// TIA Portal V20 export
FUNCTION "Safety Door" : Void   // FC97, LAD
// stored: SetENOAutomatically false
   VAR CONSTANT
      TRUE : Bool := TRUE;
      FALSE : Bool;
   END_VAR
   VAR_TEMP   // added for the SCL form of the ladder/FBD networks
      _w1 : Bool;
   END_VAR
BEGIN

REGION Network 1: FDoorEC.TOP Monitoring
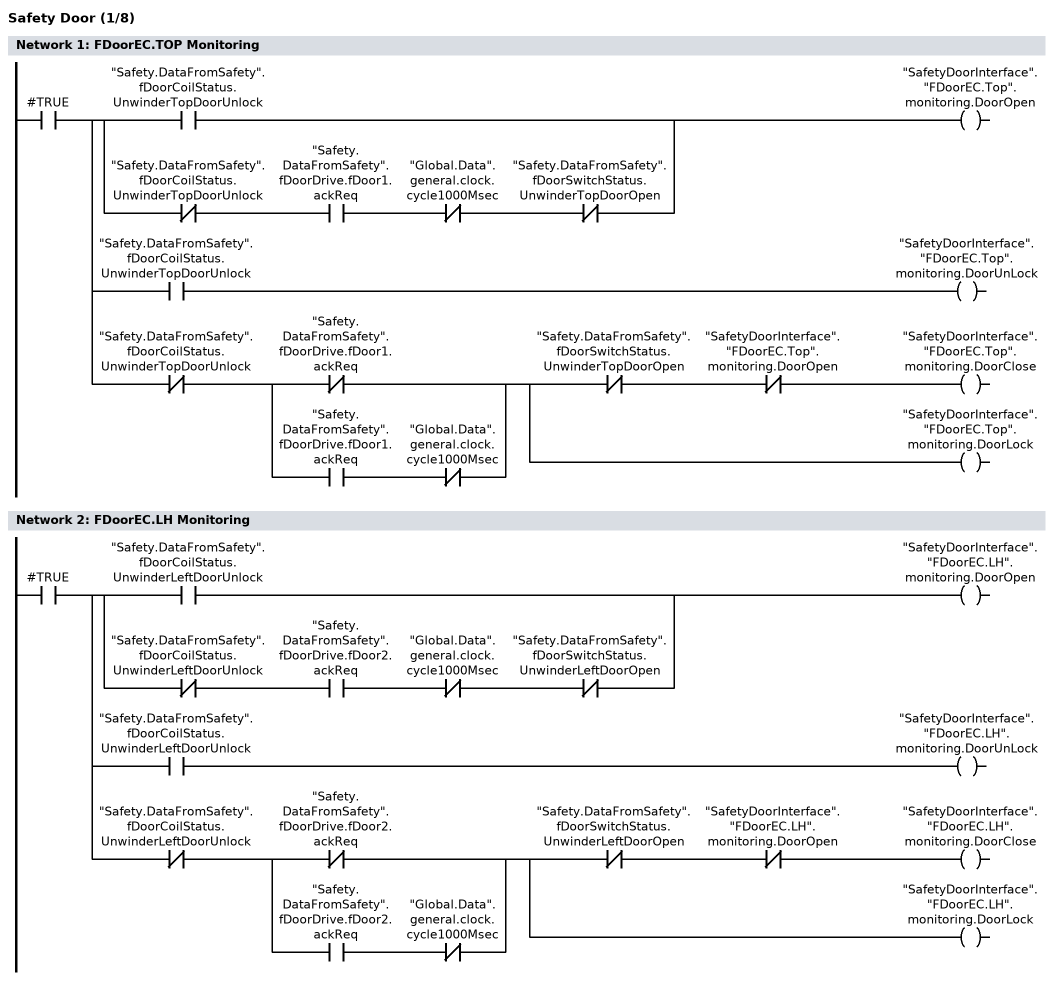
   RUNG wire#powerrail
      Contact( #TRUE )
      wire#w1
      Contact( "Safety.DataFromSafety".fDoorCoilStatus.UnwinderTopDoorUnlock )
      wire#w2
      Coil( "SafetyDoorInterface"."FDoorEC.Top".monitoring.DoorOpen )
   END_RUNG
   RUNG wire#w1
      I_Contact( "Safety.DataFromSafety".fDoorCoilStatus.UnwinderTopDoorUnlock )
      Contact( "Safety.DataFromSafety".fDoorDrive.fDoor1.ackReq )
      I_Contact( "Global.Data".general.clock.cycle1000Msec )
      I_Contact( "Safety.DataFromSafety".fDoorSwitchStatus.UnwinderTopDoorOpen )
   END_RUNG wire#w2
   RUNG wire#w1
      Contact( "Safety.DataFromSafety".fDoorCoilStatus.UnwinderTopDoorUnlock )
      Coil( "SafetyDoorInterface"."FDoorEC.Top".monitoring.DoorUnLock )
   END_RUNG
   RUNG wire#w1
      I_Contact( "Safety.DataFromSafety".fDoorCoilStatus.UnwinderTopDoorUnlock )
      wire#w3
      I_Contact( "Safety.DataFromSafety".fDoorDrive.fDoor1.ackReq )
      wire#w4
      I_Contact( "Safety.DataFromSafety".fDoorSwitchStatus.UnwinderTopDoorOpen )
      I_Contact( "SafetyDoorInterface"."FDoorEC.Top".monitoring.DoorOpen )
      Coil( "SafetyDoorInterface"."FDoorEC.Top".monitoring.DoorClose )
   END_RUNG
   RUNG wire#w3
      Contact( "Safety.DataFromSafety".fDoorDrive.fDoor1.ackReq )
      I_Contact( "Global.Data".general.clock.cycle1000Msec )
   END_RUNG wire#w4
   RUNG wire#w4
      Coil( "SafetyDoorInterface"."FDoorEC.Top".monitoring.DoorLock )
   END_RUNG
   // the same network as SCL:
   "SafetyDoorInterface"."FDoorEC.Top".monitoring.DoorOpen := #TRUE AND ("Safety.DataFromSafety".fDoorCoilStatus.UnwinderTopDoorUnlock OR (NOT "Safety.DataFromSafety".fDoorCoilStatus.UnwinderTopDoorUnlock AND "Safety.DataFromSafety".fDoorDrive.fDoor1.ackReq AND NOT "Global.Data".general.clock.cycle1000Msec AND NOT "Safety.DataFromSafety".fDoorSwitchStatus.UnwinderTopDoorOpen));
   "SafetyDoorInterface"."FDoorEC.Top".monitoring.DoorUnLock := #TRUE AND "Safety.DataFromSafety".fDoorCoilStatus.UnwinderTopDoorUnlock;
   #_w1 := #TRUE AND NOT "Safety.DataFromSafety".fDoorCoilStatus.UnwinderTopDoorUnlock AND (NOT "Safety.DataFromSafety".fDoorDrive.fDoor1.ackReq OR ("Safety.DataFromSafety".fDoorDrive.fDoor1.ackReq AND NOT "Global.Data".general.clock.cycle1000Msec));
   "SafetyDoorInterface"."FDoorEC.Top".monitoring.DoorClose := #_w1 AND NOT "Safety.DataFromSafety".fDoorSwitchStatus.UnwinderTopDoorOpen AND NOT "SafetyDoorInterface"."FDoorEC.Top".monitoring.DoorOpen;
   "SafetyDoorInterface"."FDoorEC.Top".monitoring.DoorLock := #_w1;
END_REGION

REGION Network 2: FDoorEC.LH Monitoring
   RUNG wire#powerrail
      Contact( #TRUE )
      wire#w1
      Contact( "Safety.DataFromSafety".fDoorCoilStatus.UnwinderLeftDoorUnlock )
      wire#w2
      Coil( "SafetyDoorInterface"."FDoorEC.LH".monitoring.DoorOpen )
   END_RUNG
   RUNG wire#w1
      I_Contact( "Safety.DataFromSafety".fDoorCoilStatus.UnwinderLeftDoorUnlock )
      Contact( "Safety.DataFromSafety".fDoorDrive.fDoor2.ackReq )
      I_Contact( "Global.Data".general.clock.cycle1000Msec )
      I_Contact( "Safety.DataFromSafety".fDoorSwitchStatus.UnwinderLeftDoorOpen )
   END_RUNG wire#w2
   RUNG wire#w1
      Contact( "Safety.DataFromSafety".fDoorCoilStatus.UnwinderLeftDoorUnlock )
      Coil( "SafetyDoorInterface"."FDoorEC.LH".monitoring.DoorUnLock )
   END_RUNG
   RUNG wire#w1
      I_Contact( "Safety.DataFromSafety".fDoorCoilStatus.UnwinderLeftDoorUnlock )
      wire#w3
      I_Contact( "Safety.DataFromSafety".fDoorDrive.fDoor2.ackReq )
      wire#w4
      I_Contact( "Safety.DataFromSafety".fDoorSwitchStatus.UnwinderLeftDoorOpen )
      I_Contact( "SafetyDoorInterface"."FDoorEC.LH".monitoring.DoorOpen )
      Coil( "SafetyDoorInterface"."FDoorEC.LH".monitoring.DoorClose )
   END_RUNG
   RUNG wire#w3
      Contact( "Safety.DataFromSafety".fDoorDrive.fDoor2.ackReq )
      I_Contact( "Global.Data".general.clock.cycle1000Msec )
   END_RUNG wire#w4
   RUNG wire#w4
      Coil( "SafetyDoorInterface"."FDoorEC.LH".monitoring.DoorLock )
   END_RUNG
   // the same network as SCL:
   "SafetyDoorInterface"."FDoorEC.LH".monitoring.DoorOpen := #TRUE AND ("Safety.DataFromSafety".fDoorCoilStatus.UnwinderLeftDoorUnlock OR (NOT "Safety.DataFromSafety".fDoorCoilStatus.UnwinderLeftDoorUnlock AND "Safety.DataFromSafety".fDoorDrive.fDoor2.ackReq AND NOT "Global.Data".general.clock.cycle1000Msec AND NOT "Safety.DataFromSafety".fDoorSwitchStatus.UnwinderLeftDoorOpen));
   "SafetyDoorInterface"."FDoorEC.LH".monitoring.DoorUnLock := #TRUE AND "Safety.DataFromSafety".fDoorCoilStatus.UnwinderLeftDoorUnlock;
   #_w1 := #TRUE AND NOT "Safety.DataFromSafety".fDoorCoilStatus.UnwinderLeftDoorUnlock AND (NOT "Safety.DataFromSafety".fDoorDrive.fDoor2.ackReq OR ("Safety.DataFromSafety".fDoorDrive.fDoor2.ackReq AND NOT "Global.Data".general.clock.cycle1000Msec));
   "SafetyDoorInterface"."FDoorEC.LH".monitoring.DoorClose := #_w1 AND NOT "Safety.DataFromSafety".fDoorSwitchStatus.UnwinderLeftDoorOpen AND NOT "SafetyDoorInterface"."FDoorEC.LH".monitoring.DoorOpen;
   "SafetyDoorInterface"."FDoorEC.LH".monitoring.DoorLock := #_w1;
END_REGION

REGION Network 3: FDoorEC.RH Monitoring
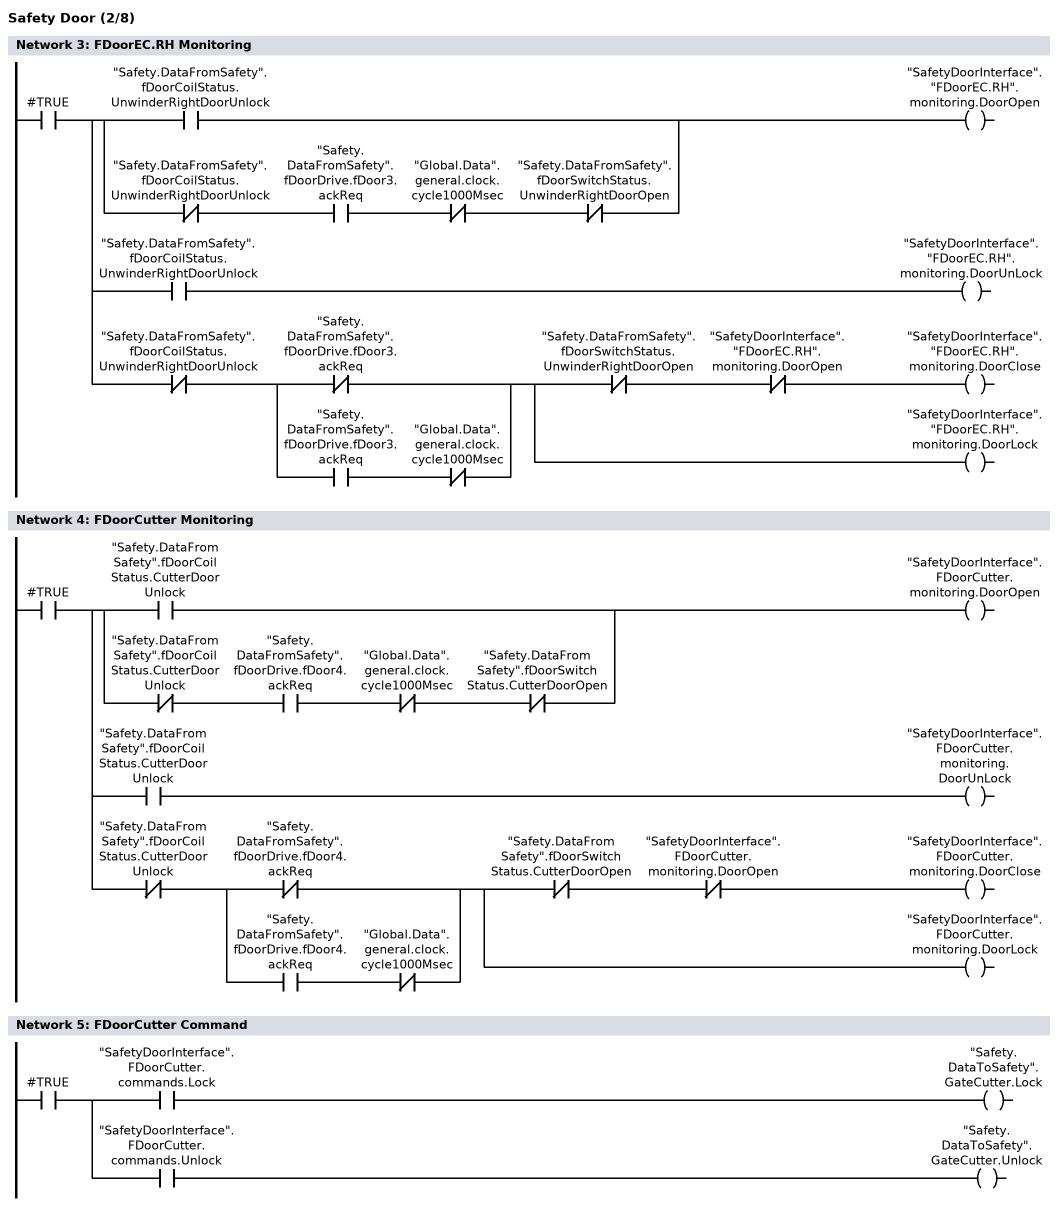
   RUNG wire#powerrail
      Contact( #TRUE )
      wire#w1
      Contact( "Safety.DataFromSafety".fDoorCoilStatus.UnwinderRightDoorUnlock )
      wire#w2
      Coil( "SafetyDoorInterface"."FDoorEC.RH".monitoring.DoorOpen )
   END_RUNG
   RUNG wire#w1
      I_Contact( "Safety.DataFromSafety".fDoorCoilStatus.UnwinderRightDoorUnlock )
      Contact( "Safety.DataFromSafety".fDoorDrive.fDoor3.ackReq )
      I_Contact( "Global.Data".general.clock.cycle1000Msec )
      I_Contact( "Safety.DataFromSafety".fDoorSwitchStatus.UnwinderRightDoorOpen )
   END_RUNG wire#w2
   RUNG wire#w1
      Contact( "Safety.DataFromSafety".fDoorCoilStatus.UnwinderRightDoorUnlock )
      Coil( "SafetyDoorInterface"."FDoorEC.RH".monitoring.DoorUnLock )
   END_RUNG
   RUNG wire#w1
      I_Contact( "Safety.DataFromSafety".fDoorCoilStatus.UnwinderRightDoorUnlock )
      wire#w3
      I_Contact( "Safety.DataFromSafety".fDoorDrive.fDoor3.ackReq )
      wire#w4
      I_Contact( "Safety.DataFromSafety".fDoorSwitchStatus.UnwinderRightDoorOpen )
      I_Contact( "SafetyDoorInterface"."FDoorEC.RH".monitoring.DoorOpen )
      Coil( "SafetyDoorInterface"."FDoorEC.RH".monitoring.DoorClose )
   END_RUNG
   RUNG wire#w3
      Contact( "Safety.DataFromSafety".fDoorDrive.fDoor3.ackReq )
      I_Contact( "Global.Data".general.clock.cycle1000Msec )
   END_RUNG wire#w4
   RUNG wire#w4
      Coil( "SafetyDoorInterface"."FDoorEC.RH".monitoring.DoorLock )
   END_RUNG
   // the same network as SCL:
   "SafetyDoorInterface"."FDoorEC.RH".monitoring.DoorOpen := #TRUE AND ("Safety.DataFromSafety".fDoorCoilStatus.UnwinderRightDoorUnlock OR (NOT "Safety.DataFromSafety".fDoorCoilStatus.UnwinderRightDoorUnlock AND "Safety.DataFromSafety".fDoorDrive.fDoor3.ackReq AND NOT "Global.Data".general.clock.cycle1000Msec AND NOT "Safety.DataFromSafety".fDoorSwitchStatus.UnwinderRightDoorOpen));
   "SafetyDoorInterface"."FDoorEC.RH".monitoring.DoorUnLock := #TRUE AND "Safety.DataFromSafety".fDoorCoilStatus.UnwinderRightDoorUnlock;
   #_w1 := #TRUE AND NOT "Safety.DataFromSafety".fDoorCoilStatus.UnwinderRightDoorUnlock AND (NOT "Safety.DataFromSafety".fDoorDrive.fDoor3.ackReq OR ("Safety.DataFromSafety".fDoorDrive.fDoor3.ackReq AND NOT "Global.Data".general.clock.cycle1000Msec));
   "SafetyDoorInterface"."FDoorEC.RH".monitoring.DoorClose := #_w1 AND NOT "Safety.DataFromSafety".fDoorSwitchStatus.UnwinderRightDoorOpen AND NOT "SafetyDoorInterface"."FDoorEC.RH".monitoring.DoorOpen;
   "SafetyDoorInterface"."FDoorEC.RH".monitoring.DoorLock := #_w1;
END_REGION

REGION Network 4: FDoorCutter Monitoring
   RUNG wire#powerrail
      Contact( #TRUE )
      wire#w1
      Contact( "Safety.DataFromSafety".fDoorCoilStatus.CutterDoorUnlock )
      wire#w2
      Coil( "SafetyDoorInterface".FDoorCutter.monitoring.DoorOpen )
   END_RUNG
   RUNG wire#w1
      I_Contact( "Safety.DataFromSafety".fDoorCoilStatus.CutterDoorUnlock )
      Contact( "Safety.DataFromSafety".fDoorDrive.fDoor4.ackReq )
      I_Contact( "Global.Data".general.clock.cycle1000Msec )
      I_Contact( "Safety.DataFromSafety".fDoorSwitchStatus.CutterDoorOpen )
   END_RUNG wire#w2
   RUNG wire#w1
      Contact( "Safety.DataFromSafety".fDoorCoilStatus.CutterDoorUnlock )
      Coil( "SafetyDoorInterface".FDoorCutter.monitoring.DoorUnLock )
   END_RUNG
   RUNG wire#w1
      I_Contact( "Safety.DataFromSafety".fDoorCoilStatus.CutterDoorUnlock )
      wire#w3
      I_Contact( "Safety.DataFromSafety".fDoorDrive.fDoor4.ackReq )
      wire#w4
      I_Contact( "Safety.DataFromSafety".fDoorSwitchStatus.CutterDoorOpen )
      I_Contact( "SafetyDoorInterface".FDoorCutter.monitoring.DoorOpen )
      Coil( "SafetyDoorInterface".FDoorCutter.monitoring.DoorClose )
   END_RUNG
   RUNG wire#w3
      Contact( "Safety.DataFromSafety".fDoorDrive.fDoor4.ackReq )
      I_Contact( "Global.Data".general.clock.cycle1000Msec )
   END_RUNG wire#w4
   RUNG wire#w4
      Coil( "SafetyDoorInterface".FDoorCutter.monitoring.DoorLock )
   END_RUNG
   // the same network as SCL:
   "SafetyDoorInterface".FDoorCutter.monitoring.DoorOpen := #TRUE AND ("Safety.DataFromSafety".fDoorCoilStatus.CutterDoorUnlock OR (NOT "Safety.DataFromSafety".fDoorCoilStatus.CutterDoorUnlock AND "Safety.DataFromSafety".fDoorDrive.fDoor4.ackReq AND NOT "Global.Data".general.clock.cycle1000Msec AND NOT "Safety.DataFromSafety".fDoorSwitchStatus.CutterDoorOpen));
   "SafetyDoorInterface".FDoorCutter.monitoring.DoorUnLock := #TRUE AND "Safety.DataFromSafety".fDoorCoilStatus.CutterDoorUnlock;
   #_w1 := #TRUE AND NOT "Safety.DataFromSafety".fDoorCoilStatus.CutterDoorUnlock AND (NOT "Safety.DataFromSafety".fDoorDrive.fDoor4.ackReq OR ("Safety.DataFromSafety".fDoorDrive.fDoor4.ackReq AND NOT "Global.Data".general.clock.cycle1000Msec));
   "SafetyDoorInterface".FDoorCutter.monitoring.DoorClose := #_w1 AND NOT "Safety.DataFromSafety".fDoorSwitchStatus.CutterDoorOpen AND NOT "SafetyDoorInterface".FDoorCutter.monitoring.DoorOpen;
   "SafetyDoorInterface".FDoorCutter.monitoring.DoorLock := #_w1;
END_REGION

REGION Network 5: FDoorCutter Command
   RUNG wire#powerrail
      Contact( #TRUE )
      wire#w1
      Contact( "SafetyDoorInterface".FDoorCutter.commands.Lock )
      Coil( "Safety.DataToSafety".GateCutter.Lock )
   END_RUNG
   RUNG wire#w1
      Contact( "SafetyDoorInterface".FDoorCutter.commands.Unlock )
      Coil( "Safety.DataToSafety".GateCutter.Unlock )
   END_RUNG
   // the same network as SCL:
   "Safety.DataToSafety".GateCutter.Lock := #TRUE AND "SafetyDoorInterface".FDoorCutter.commands.Lock;
   "Safety.DataToSafety".GateCutter.Unlock := #TRUE AND "SafetyDoorInterface".FDoorCutter.commands.Unlock;
END_REGION

REGION Network 6: FDoorMagazine Monitoring
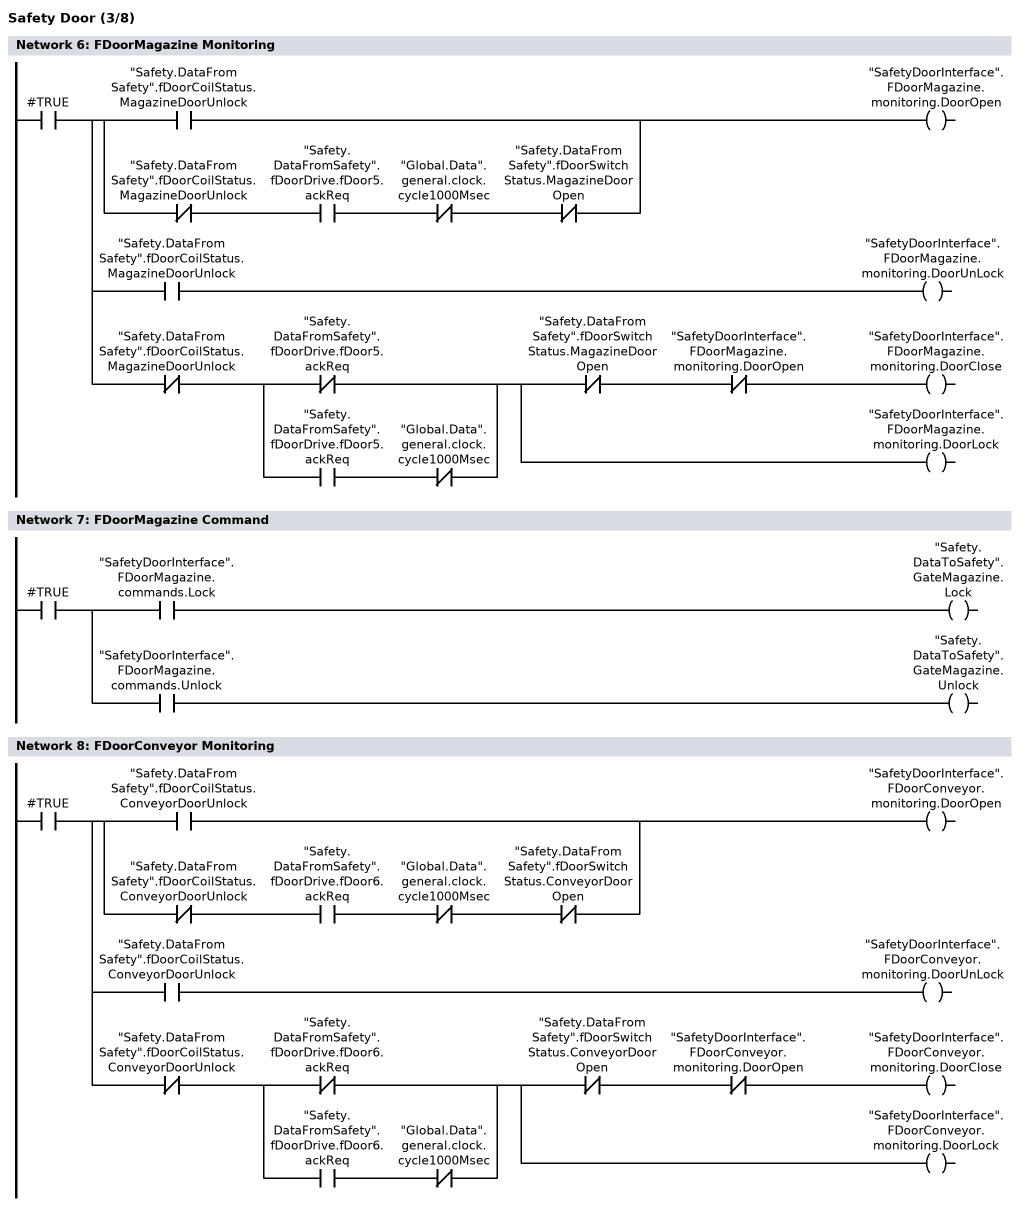
   RUNG wire#powerrail
      Contact( #TRUE )
      wire#w1
      Contact( "Safety.DataFromSafety".fDoorCoilStatus.MagazineDoorUnlock )
      wire#w2
      Coil( "SafetyDoorInterface".FDoorMagazine.monitoring.DoorOpen )
   END_RUNG
   RUNG wire#w1
      I_Contact( "Safety.DataFromSafety".fDoorCoilStatus.MagazineDoorUnlock )
      Contact( "Safety.DataFromSafety".fDoorDrive.fDoor5.ackReq )
      I_Contact( "Global.Data".general.clock.cycle1000Msec )
      I_Contact( "Safety.DataFromSafety".fDoorSwitchStatus.MagazineDoorOpen )
   END_RUNG wire#w2
   RUNG wire#w1
      Contact( "Safety.DataFromSafety".fDoorCoilStatus.MagazineDoorUnlock )
      Coil( "SafetyDoorInterface".FDoorMagazine.monitoring.DoorUnLock )
   END_RUNG
   RUNG wire#w1
      I_Contact( "Safety.DataFromSafety".fDoorCoilStatus.MagazineDoorUnlock )
      wire#w3
      I_Contact( "Safety.DataFromSafety".fDoorDrive.fDoor5.ackReq )
      wire#w4
      I_Contact( "Safety.DataFromSafety".fDoorSwitchStatus.MagazineDoorOpen )
      I_Contact( "SafetyDoorInterface".FDoorMagazine.monitoring.DoorOpen )
      Coil( "SafetyDoorInterface".FDoorMagazine.monitoring.DoorClose )
   END_RUNG
   RUNG wire#w3
      Contact( "Safety.DataFromSafety".fDoorDrive.fDoor5.ackReq )
      I_Contact( "Global.Data".general.clock.cycle1000Msec )
   END_RUNG wire#w4
   RUNG wire#w4
      Coil( "SafetyDoorInterface".FDoorMagazine.monitoring.DoorLock )
   END_RUNG
   // the same network as SCL:
   "SafetyDoorInterface".FDoorMagazine.monitoring.DoorOpen := #TRUE AND ("Safety.DataFromSafety".fDoorCoilStatus.MagazineDoorUnlock OR (NOT "Safety.DataFromSafety".fDoorCoilStatus.MagazineDoorUnlock AND "Safety.DataFromSafety".fDoorDrive.fDoor5.ackReq AND NOT "Global.Data".general.clock.cycle1000Msec AND NOT "Safety.DataFromSafety".fDoorSwitchStatus.MagazineDoorOpen));
   "SafetyDoorInterface".FDoorMagazine.monitoring.DoorUnLock := #TRUE AND "Safety.DataFromSafety".fDoorCoilStatus.MagazineDoorUnlock;
   #_w1 := #TRUE AND NOT "Safety.DataFromSafety".fDoorCoilStatus.MagazineDoorUnlock AND (NOT "Safety.DataFromSafety".fDoorDrive.fDoor5.ackReq OR ("Safety.DataFromSafety".fDoorDrive.fDoor5.ackReq AND NOT "Global.Data".general.clock.cycle1000Msec));
   "SafetyDoorInterface".FDoorMagazine.monitoring.DoorClose := #_w1 AND NOT "Safety.DataFromSafety".fDoorSwitchStatus.MagazineDoorOpen AND NOT "SafetyDoorInterface".FDoorMagazine.monitoring.DoorOpen;
   "SafetyDoorInterface".FDoorMagazine.monitoring.DoorLock := #_w1;
END_REGION

REGION Network 7: FDoorMagazine Command
   RUNG wire#powerrail
      Contact( #TRUE )
      wire#w1
      Contact( "SafetyDoorInterface".FDoorMagazine.commands.Lock )
      Coil( "Safety.DataToSafety".GateMagazine.Lock )
   END_RUNG
   RUNG wire#w1
      Contact( "SafetyDoorInterface".FDoorMagazine.commands.Unlock )
      Coil( "Safety.DataToSafety".GateMagazine.Unlock )
   END_RUNG
   // the same network as SCL:
   "Safety.DataToSafety".GateMagazine.Lock := #TRUE AND "SafetyDoorInterface".FDoorMagazine.commands.Lock;
   "Safety.DataToSafety".GateMagazine.Unlock := #TRUE AND "SafetyDoorInterface".FDoorMagazine.commands.Unlock;
END_REGION

REGION Network 8: FDoorConveyor Monitoring
   RUNG wire#powerrail
      Contact( #TRUE )
      wire#w1
      Contact( "Safety.DataFromSafety".fDoorCoilStatus.ConveyorDoorUnlock )
      wire#w2
      Coil( "SafetyDoorInterface".FDoorConveyor.monitoring.DoorOpen )
   END_RUNG
   RUNG wire#w1
      I_Contact( "Safety.DataFromSafety".fDoorCoilStatus.ConveyorDoorUnlock )
      Contact( "Safety.DataFromSafety".fDoorDrive.fDoor6.ackReq )
      I_Contact( "Global.Data".general.clock.cycle1000Msec )
      I_Contact( "Safety.DataFromSafety".fDoorSwitchStatus.ConveyorDoorOpen )
   END_RUNG wire#w2
   RUNG wire#w1
      Contact( "Safety.DataFromSafety".fDoorCoilStatus.ConveyorDoorUnlock )
      Coil( "SafetyDoorInterface".FDoorConveyor.monitoring.DoorUnLock )
   END_RUNG
   RUNG wire#w1
      I_Contact( "Safety.DataFromSafety".fDoorCoilStatus.ConveyorDoorUnlock )
      wire#w3
      I_Contact( "Safety.DataFromSafety".fDoorDrive.fDoor6.ackReq )
      wire#w4
      I_Contact( "Safety.DataFromSafety".fDoorSwitchStatus.ConveyorDoorOpen )
      I_Contact( "SafetyDoorInterface".FDoorConveyor.monitoring.DoorOpen )
      Coil( "SafetyDoorInterface".FDoorConveyor.monitoring.DoorClose )
   END_RUNG
   RUNG wire#w3
      Contact( "Safety.DataFromSafety".fDoorDrive.fDoor6.ackReq )
      I_Contact( "Global.Data".general.clock.cycle1000Msec )
   END_RUNG wire#w4
   RUNG wire#w4
      Coil( "SafetyDoorInterface".FDoorConveyor.monitoring.DoorLock )
   END_RUNG
   // the same network as SCL:
   "SafetyDoorInterface".FDoorConveyor.monitoring.DoorOpen := #TRUE AND ("Safety.DataFromSafety".fDoorCoilStatus.ConveyorDoorUnlock OR (NOT "Safety.DataFromSafety".fDoorCoilStatus.ConveyorDoorUnlock AND "Safety.DataFromSafety".fDoorDrive.fDoor6.ackReq AND NOT "Global.Data".general.clock.cycle1000Msec AND NOT "Safety.DataFromSafety".fDoorSwitchStatus.ConveyorDoorOpen));
   "SafetyDoorInterface".FDoorConveyor.monitoring.DoorUnLock := #TRUE AND "Safety.DataFromSafety".fDoorCoilStatus.ConveyorDoorUnlock;
   #_w1 := #TRUE AND NOT "Safety.DataFromSafety".fDoorCoilStatus.ConveyorDoorUnlock AND (NOT "Safety.DataFromSafety".fDoorDrive.fDoor6.ackReq OR ("Safety.DataFromSafety".fDoorDrive.fDoor6.ackReq AND NOT "Global.Data".general.clock.cycle1000Msec));
   "SafetyDoorInterface".FDoorConveyor.monitoring.DoorClose := #_w1 AND NOT "Safety.DataFromSafety".fDoorSwitchStatus.ConveyorDoorOpen AND NOT "SafetyDoorInterface".FDoorConveyor.monitoring.DoorOpen;
   "SafetyDoorInterface".FDoorConveyor.monitoring.DoorLock := #_w1;
END_REGION

REGION Network 9: FDoorConveyor Command
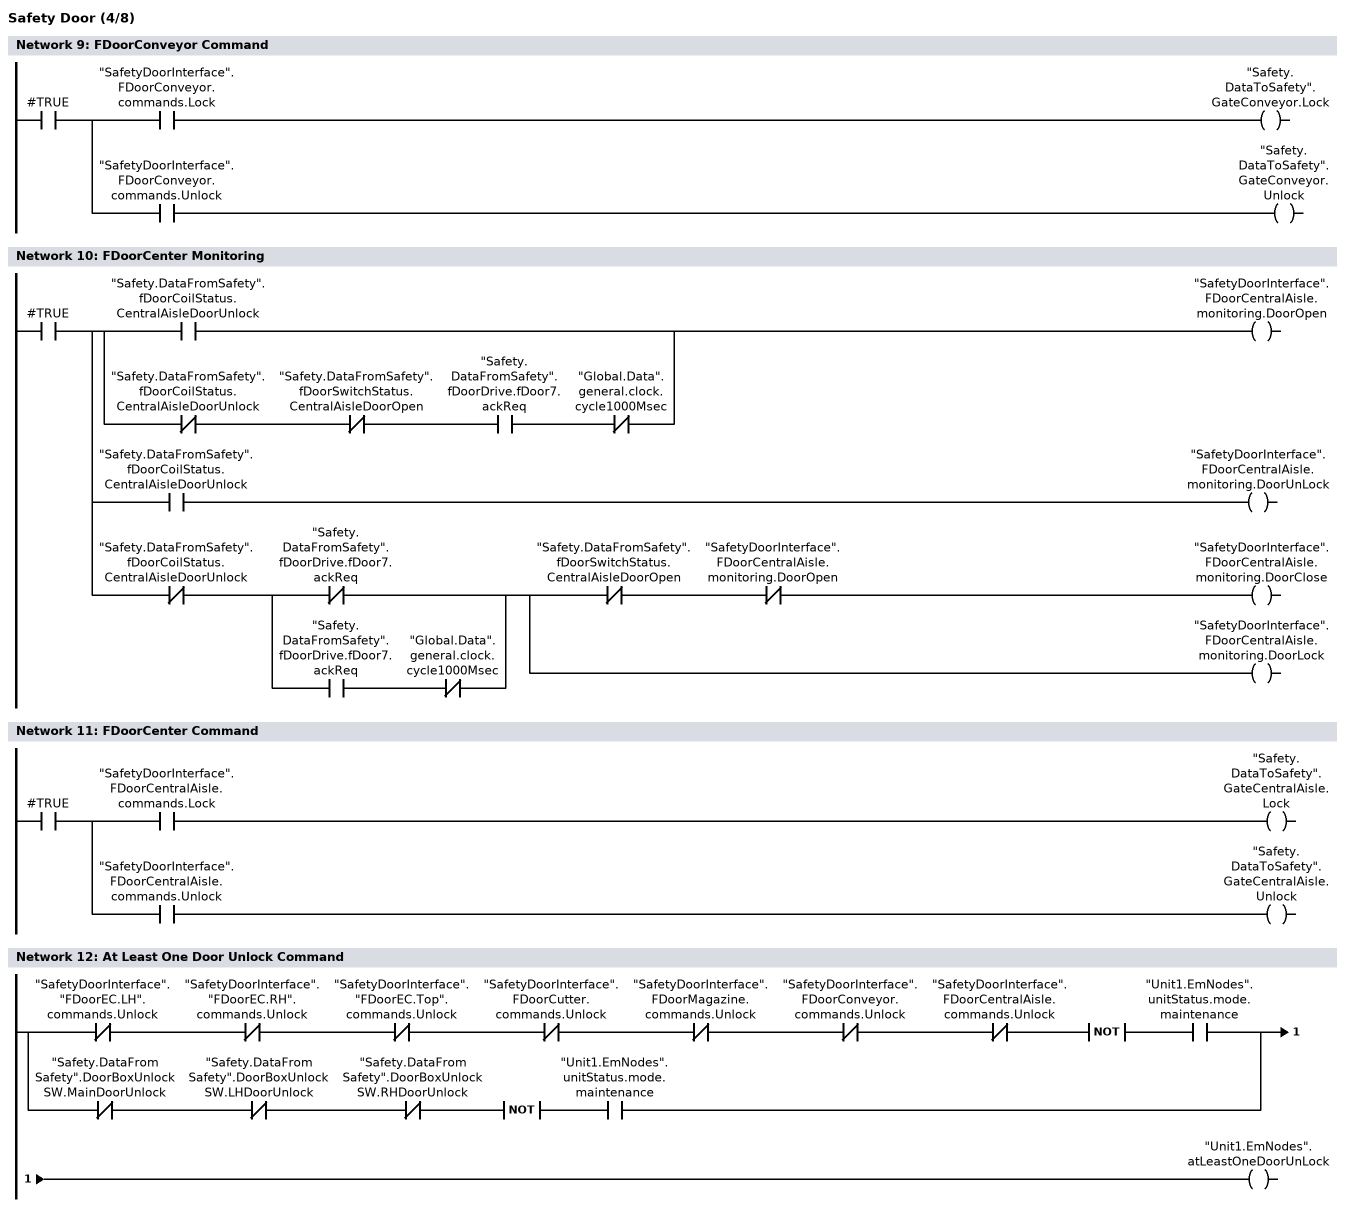
   RUNG wire#powerrail
      Contact( #TRUE )
      wire#w1
      Contact( "SafetyDoorInterface".FDoorConveyor.commands.Lock )
      Coil( "Safety.DataToSafety".GateConveyor.Lock )
   END_RUNG
   RUNG wire#w1
      Contact( "SafetyDoorInterface".FDoorConveyor.commands.Unlock )
      Coil( "Safety.DataToSafety".GateConveyor.Unlock )
   END_RUNG
   // the same network as SCL:
   "Safety.DataToSafety".GateConveyor.Lock := #TRUE AND "SafetyDoorInterface".FDoorConveyor.commands.Lock;
   "Safety.DataToSafety".GateConveyor.Unlock := #TRUE AND "SafetyDoorInterface".FDoorConveyor.commands.Unlock;
END_REGION

REGION Network 10: FDoorCenter Monitoring
   RUNG wire#powerrail
      Contact( #TRUE )
      wire#w1
      Contact( "Safety.DataFromSafety".fDoorCoilStatus.CentralAisleDoorUnlock )
      wire#w2
      Coil( "SafetyDoorInterface".FDoorCentralAisle.monitoring.DoorOpen )
   END_RUNG
   RUNG wire#w1
      I_Contact( "Safety.DataFromSafety".fDoorCoilStatus.CentralAisleDoorUnlock )
      I_Contact( "Safety.DataFromSafety".fDoorSwitchStatus.CentralAisleDoorOpen )
      Contact( "Safety.DataFromSafety".fDoorDrive.fDoor7.ackReq )
      I_Contact( "Global.Data".general.clock.cycle1000Msec )
   END_RUNG wire#w2
   RUNG wire#w1
      Contact( "Safety.DataFromSafety".fDoorCoilStatus.CentralAisleDoorUnlock )
      Coil( "SafetyDoorInterface".FDoorCentralAisle.monitoring.DoorUnLock )
   END_RUNG
   RUNG wire#w1
      I_Contact( "Safety.DataFromSafety".fDoorCoilStatus.CentralAisleDoorUnlock )
      wire#w3
      I_Contact( "Safety.DataFromSafety".fDoorDrive.fDoor7.ackReq )
      wire#w4
      I_Contact( "Safety.DataFromSafety".fDoorSwitchStatus.CentralAisleDoorOpen )
      I_Contact( "SafetyDoorInterface".FDoorCentralAisle.monitoring.DoorOpen )
      Coil( "SafetyDoorInterface".FDoorCentralAisle.monitoring.DoorClose )
   END_RUNG
   RUNG wire#w3
      Contact( "Safety.DataFromSafety".fDoorDrive.fDoor7.ackReq )
      I_Contact( "Global.Data".general.clock.cycle1000Msec )
   END_RUNG wire#w4
   RUNG wire#w4
      Coil( "SafetyDoorInterface".FDoorCentralAisle.monitoring.DoorLock )
   END_RUNG
   // the same network as SCL:
   "SafetyDoorInterface".FDoorCentralAisle.monitoring.DoorOpen := #TRUE AND ("Safety.DataFromSafety".fDoorCoilStatus.CentralAisleDoorUnlock OR (NOT "Safety.DataFromSafety".fDoorCoilStatus.CentralAisleDoorUnlock AND NOT "Safety.DataFromSafety".fDoorSwitchStatus.CentralAisleDoorOpen AND "Safety.DataFromSafety".fDoorDrive.fDoor7.ackReq AND NOT "Global.Data".general.clock.cycle1000Msec));
   "SafetyDoorInterface".FDoorCentralAisle.monitoring.DoorUnLock := #TRUE AND "Safety.DataFromSafety".fDoorCoilStatus.CentralAisleDoorUnlock;
   #_w1 := #TRUE AND NOT "Safety.DataFromSafety".fDoorCoilStatus.CentralAisleDoorUnlock AND (NOT "Safety.DataFromSafety".fDoorDrive.fDoor7.ackReq OR ("Safety.DataFromSafety".fDoorDrive.fDoor7.ackReq AND NOT "Global.Data".general.clock.cycle1000Msec));
   "SafetyDoorInterface".FDoorCentralAisle.monitoring.DoorClose := #_w1 AND NOT "Safety.DataFromSafety".fDoorSwitchStatus.CentralAisleDoorOpen AND NOT "SafetyDoorInterface".FDoorCentralAisle.monitoring.DoorOpen;
   "SafetyDoorInterface".FDoorCentralAisle.monitoring.DoorLock := #_w1;
END_REGION

REGION Network 11: FDoorCenter Command
   RUNG wire#powerrail
      Contact( #TRUE )
      wire#w1
      Contact( "SafetyDoorInterface".FDoorCentralAisle.commands.Lock )
      Coil( "Safety.DataToSafety".GateCentralAisle.Lock )
   END_RUNG
   RUNG wire#w1
      Contact( "SafetyDoorInterface".FDoorCentralAisle.commands.Unlock )
      Coil( "Safety.DataToSafety".GateCentralAisle.Unlock )
   END_RUNG
   // the same network as SCL:
   "Safety.DataToSafety".GateCentralAisle.Lock := #TRUE AND "SafetyDoorInterface".FDoorCentralAisle.commands.Lock;
   "Safety.DataToSafety".GateCentralAisle.Unlock := #TRUE AND "SafetyDoorInterface".FDoorCentralAisle.commands.Unlock;
END_REGION

REGION Network 12: At Least One Door Unlock Command
   RUNG wire#powerrail
      I_Contact( "SafetyDoorInterface"."FDoorEC.LH".commands.Unlock )
      I_Contact( "SafetyDoorInterface"."FDoorEC.RH".commands.Unlock )
      I_Contact( "SafetyDoorInterface"."FDoorEC.Top".commands.Unlock )
      I_Contact( "SafetyDoorInterface".FDoorCutter.commands.Unlock )
      I_Contact( "SafetyDoorInterface".FDoorMagazine.commands.Unlock )
      I_Contact( "SafetyDoorInterface".FDoorConveyor.commands.Unlock )
      I_Contact( "SafetyDoorInterface".FDoorCentralAisle.commands.Unlock )
      Not()
      Contact( "Unit1.EmNodes".unitStatus.mode.maintenance )
      wire#w1
      Coil( "Unit1.EmNodes".atLeastOneDoorUnLock )
   END_RUNG
   RUNG wire#powerrail
      I_Contact( "Safety.DataFromSafety".DoorBoxUnlockSW.MainDoorUnlock )
      I_Contact( "Safety.DataFromSafety".DoorBoxUnlockSW.LHDoorUnlock )
      I_Contact( "Safety.DataFromSafety".DoorBoxUnlockSW.RHDoorUnlock )
      Not()
      Contact( "Unit1.EmNodes".unitStatus.mode.maintenance )
   END_RUNG wire#w1
   // the same network as SCL:
   "Unit1.EmNodes".atLeastOneDoorUnLock := (NOT (NOT "SafetyDoorInterface"."FDoorEC.LH".commands.Unlock AND NOT "SafetyDoorInterface"."FDoorEC.RH".commands.Unlock AND NOT "SafetyDoorInterface"."FDoorEC.Top".commands.Unlock AND NOT "SafetyDoorInterface".FDoorCutter.commands.Unlock AND NOT "SafetyDoorInterface".FDoorMagazine.commands.Unlock AND NOT "SafetyDoorInterface".FDoorConveyor.commands.Unlock AND NOT "SafetyDoorInterface".FDoorCentralAisle.commands.Unlock) AND "Unit1.EmNodes".unitStatus.mode.maintenance) OR (NOT (NOT "Safety.DataFromSafety".DoorBoxUnlockSW.MainDoorUnlock AND NOT "Safety.DataFromSafety".DoorBoxUnlockSW.LHDoorUnlock AND NOT "Safety.DataFromSafety".DoorBoxUnlockSW.RHDoorUnlock) AND "Unit1.EmNodes".unitStatus.mode.maintenance);
END_REGION

REGION Network 13: OtherDoor1 Monitoring - BA015
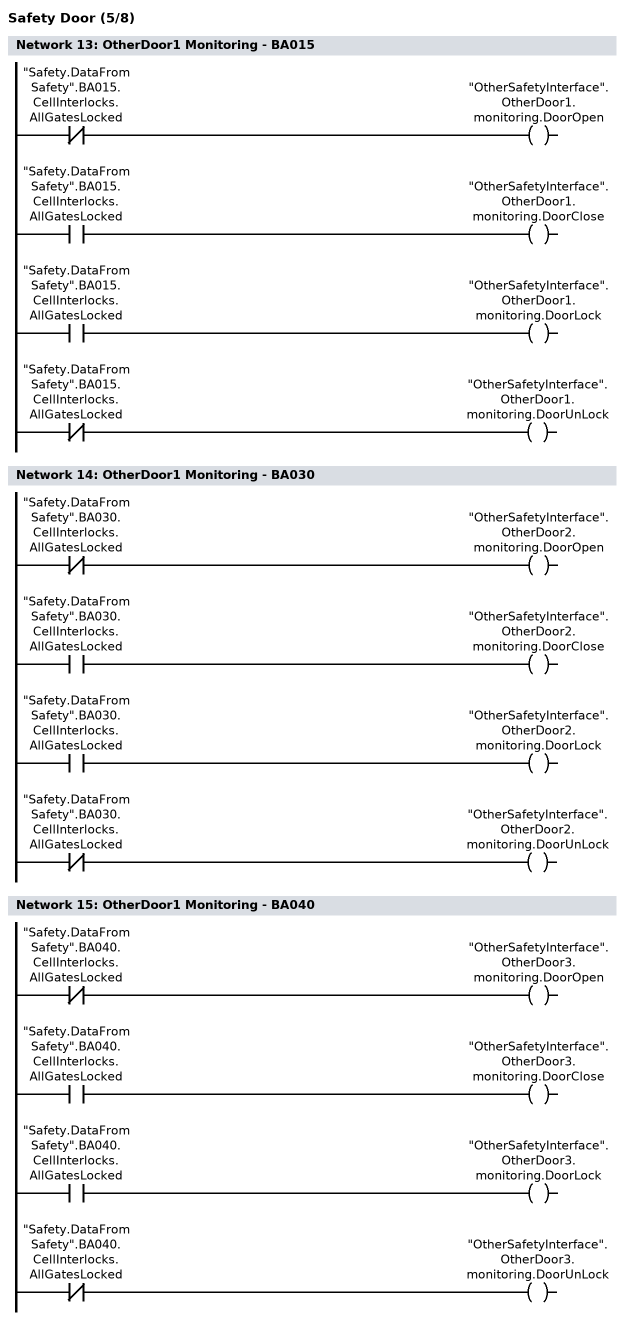
   RUNG wire#powerrail
      I_Contact( "Safety.DataFromSafety".BA015.CellInterlocks.AllGatesLocked )
      Coil( "OtherSafetyInterface".OtherDoor1.monitoring.DoorOpen )
   END_RUNG
   RUNG wire#powerrail
      Contact( "Safety.DataFromSafety".BA015.CellInterlocks.AllGatesLocked )
      Coil( "OtherSafetyInterface".OtherDoor1.monitoring.DoorClose )
   END_RUNG
   RUNG wire#powerrail
      Contact( "Safety.DataFromSafety".BA015.CellInterlocks.AllGatesLocked )
      Coil( "OtherSafetyInterface".OtherDoor1.monitoring.DoorLock )
   END_RUNG
   RUNG wire#powerrail
      I_Contact( "Safety.DataFromSafety".BA015.CellInterlocks.AllGatesLocked )
      Coil( "OtherSafetyInterface".OtherDoor1.monitoring.DoorUnLock )
   END_RUNG
   // the same network as SCL:
   "OtherSafetyInterface".OtherDoor1.monitoring.DoorOpen := NOT "Safety.DataFromSafety".BA015.CellInterlocks.AllGatesLocked;
   "OtherSafetyInterface".OtherDoor1.monitoring.DoorClose := "Safety.DataFromSafety".BA015.CellInterlocks.AllGatesLocked;
   "OtherSafetyInterface".OtherDoor1.monitoring.DoorLock := "Safety.DataFromSafety".BA015.CellInterlocks.AllGatesLocked;
   "OtherSafetyInterface".OtherDoor1.monitoring.DoorUnLock := NOT "Safety.DataFromSafety".BA015.CellInterlocks.AllGatesLocked;
END_REGION

REGION Network 14: OtherDoor1 Monitoring - BA030
   RUNG wire#powerrail
      I_Contact( "Safety.DataFromSafety".BA030.CellInterlocks.AllGatesLocked )
      Coil( "OtherSafetyInterface".OtherDoor2.monitoring.DoorOpen )
   END_RUNG
   RUNG wire#powerrail
      Contact( "Safety.DataFromSafety".BA030.CellInterlocks.AllGatesLocked )
      Coil( "OtherSafetyInterface".OtherDoor2.monitoring.DoorClose )
   END_RUNG
   RUNG wire#powerrail
      Contact( "Safety.DataFromSafety".BA030.CellInterlocks.AllGatesLocked )
      Coil( "OtherSafetyInterface".OtherDoor2.monitoring.DoorLock )
   END_RUNG
   RUNG wire#powerrail
      I_Contact( "Safety.DataFromSafety".BA030.CellInterlocks.AllGatesLocked )
      Coil( "OtherSafetyInterface".OtherDoor2.monitoring.DoorUnLock )
   END_RUNG
   // the same network as SCL:
   "OtherSafetyInterface".OtherDoor2.monitoring.DoorOpen := NOT "Safety.DataFromSafety".BA030.CellInterlocks.AllGatesLocked;
   "OtherSafetyInterface".OtherDoor2.monitoring.DoorClose := "Safety.DataFromSafety".BA030.CellInterlocks.AllGatesLocked;
   "OtherSafetyInterface".OtherDoor2.monitoring.DoorLock := "Safety.DataFromSafety".BA030.CellInterlocks.AllGatesLocked;
   "OtherSafetyInterface".OtherDoor2.monitoring.DoorUnLock := NOT "Safety.DataFromSafety".BA030.CellInterlocks.AllGatesLocked;
END_REGION

REGION Network 15: OtherDoor1 Monitoring - BA040
   RUNG wire#powerrail
      I_Contact( "Safety.DataFromSafety".BA040.CellInterlocks.AllGatesLocked )
      Coil( "OtherSafetyInterface".OtherDoor3.monitoring.DoorOpen )
   END_RUNG
   RUNG wire#powerrail
      Contact( "Safety.DataFromSafety".BA040.CellInterlocks.AllGatesLocked )
      Coil( "OtherSafetyInterface".OtherDoor3.monitoring.DoorClose )
   END_RUNG
   RUNG wire#powerrail
      Contact( "Safety.DataFromSafety".BA040.CellInterlocks.AllGatesLocked )
      Coil( "OtherSafetyInterface".OtherDoor3.monitoring.DoorLock )
   END_RUNG
   RUNG wire#powerrail
      I_Contact( "Safety.DataFromSafety".BA040.CellInterlocks.AllGatesLocked )
      Coil( "OtherSafetyInterface".OtherDoor3.monitoring.DoorUnLock )
   END_RUNG
   // the same network as SCL:
   "OtherSafetyInterface".OtherDoor3.monitoring.DoorOpen := NOT "Safety.DataFromSafety".BA040.CellInterlocks.AllGatesLocked;
   "OtherSafetyInterface".OtherDoor3.monitoring.DoorClose := "Safety.DataFromSafety".BA040.CellInterlocks.AllGatesLocked;
   "OtherSafetyInterface".OtherDoor3.monitoring.DoorLock := "Safety.DataFromSafety".BA040.CellInterlocks.AllGatesLocked;
   "OtherSafetyInterface".OtherDoor3.monitoring.DoorUnLock := NOT "Safety.DataFromSafety".BA040.CellInterlocks.AllGatesLocked;
END_REGION

REGION Network 16: OtherDoor1 Monitoring - BA060
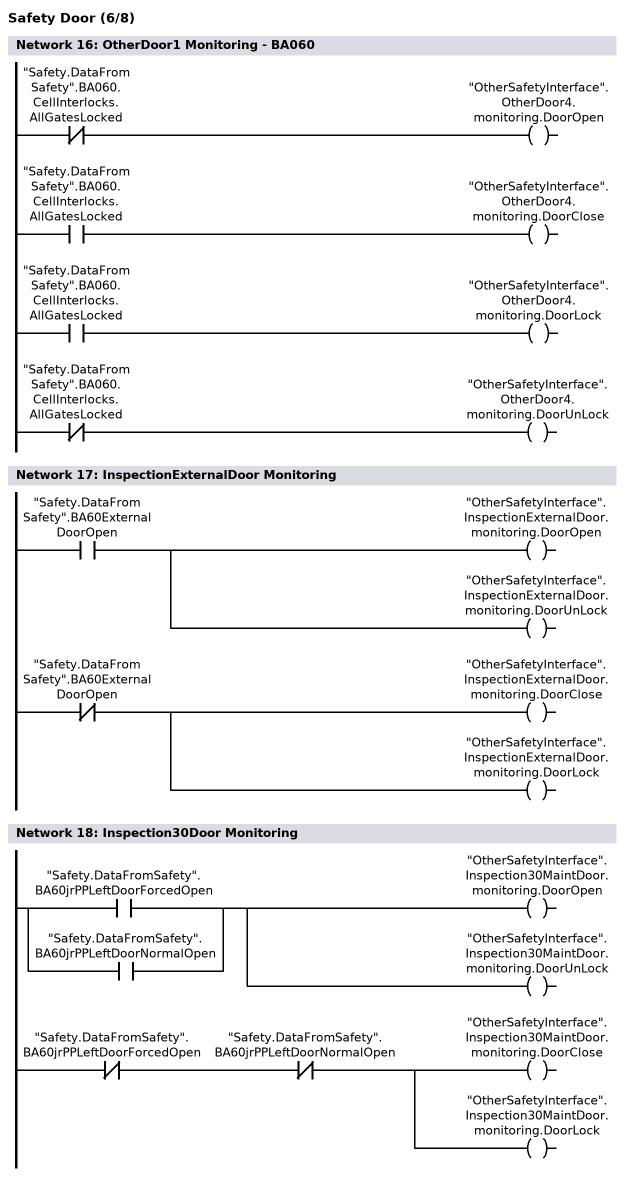
   RUNG wire#powerrail
      I_Contact( "Safety.DataFromSafety".BA060.CellInterlocks.AllGatesLocked )
      Coil( "OtherSafetyInterface".OtherDoor4.monitoring.DoorOpen )
   END_RUNG
   RUNG wire#powerrail
      Contact( "Safety.DataFromSafety".BA060.CellInterlocks.AllGatesLocked )
      Coil( "OtherSafetyInterface".OtherDoor4.monitoring.DoorClose )
   END_RUNG
   RUNG wire#powerrail
      Contact( "Safety.DataFromSafety".BA060.CellInterlocks.AllGatesLocked )
      Coil( "OtherSafetyInterface".OtherDoor4.monitoring.DoorLock )
   END_RUNG
   RUNG wire#powerrail
      I_Contact( "Safety.DataFromSafety".BA060.CellInterlocks.AllGatesLocked )
      Coil( "OtherSafetyInterface".OtherDoor4.monitoring.DoorUnLock )
   END_RUNG
   // the same network as SCL:
   "OtherSafetyInterface".OtherDoor4.monitoring.DoorOpen := NOT "Safety.DataFromSafety".BA060.CellInterlocks.AllGatesLocked;
   "OtherSafetyInterface".OtherDoor4.monitoring.DoorClose := "Safety.DataFromSafety".BA060.CellInterlocks.AllGatesLocked;
   "OtherSafetyInterface".OtherDoor4.monitoring.DoorLock := "Safety.DataFromSafety".BA060.CellInterlocks.AllGatesLocked;
   "OtherSafetyInterface".OtherDoor4.monitoring.DoorUnLock := NOT "Safety.DataFromSafety".BA060.CellInterlocks.AllGatesLocked;
END_REGION

REGION Network 17: InspectionExternalDoor Monitoring
   RUNG wire#powerrail
      Contact( "Safety.DataFromSafety".BA60ExternalDoorOpen )
      wire#w1
      Coil( "OtherSafetyInterface".InspectionExternalDoor.monitoring.DoorOpen )
   END_RUNG
   RUNG wire#w1
      Coil( "OtherSafetyInterface".InspectionExternalDoor.monitoring.DoorUnLock )
   END_RUNG
   RUNG wire#powerrail
      I_Contact( "Safety.DataFromSafety".BA60ExternalDoorOpen )
      wire#w2
      Coil( "OtherSafetyInterface".InspectionExternalDoor.monitoring.DoorClose )
   END_RUNG
   RUNG wire#w2
      Coil( "OtherSafetyInterface".InspectionExternalDoor.monitoring.DoorLock )
   END_RUNG
   // the same network as SCL:
   "OtherSafetyInterface".InspectionExternalDoor.monitoring.DoorOpen := "Safety.DataFromSafety".BA60ExternalDoorOpen;
   "OtherSafetyInterface".InspectionExternalDoor.monitoring.DoorUnLock := "Safety.DataFromSafety".BA60ExternalDoorOpen;
   "OtherSafetyInterface".InspectionExternalDoor.monitoring.DoorClose := NOT "Safety.DataFromSafety".BA60ExternalDoorOpen;
   "OtherSafetyInterface".InspectionExternalDoor.monitoring.DoorLock := NOT "Safety.DataFromSafety".BA60ExternalDoorOpen;
END_REGION

REGION Network 18: Inspection30Door Monitoring
   RUNG wire#powerrail
      Contact( "Safety.DataFromSafety".BA60jrPPLeftDoorForcedOpen )
      wire#w1
      Coil( "OtherSafetyInterface".Inspection30MaintDoor.monitoring.DoorOpen )
   END_RUNG
   RUNG wire#powerrail
      Contact( "Safety.DataFromSafety".BA60jrPPLeftDoorNormalOpen )
   END_RUNG wire#w1
   RUNG wire#w1
      Coil( "OtherSafetyInterface".Inspection30MaintDoor.monitoring.DoorUnLock )
   END_RUNG
   RUNG wire#powerrail
      I_Contact( "Safety.DataFromSafety".BA60jrPPLeftDoorForcedOpen )
      I_Contact( "Safety.DataFromSafety".BA60jrPPLeftDoorNormalOpen )
      wire#w2
      Coil( "OtherSafetyInterface".Inspection30MaintDoor.monitoring.DoorClose )
   END_RUNG
   RUNG wire#w2
      Coil( "OtherSafetyInterface".Inspection30MaintDoor.monitoring.DoorLock )
   END_RUNG
   // the same network as SCL:
   "OtherSafetyInterface".Inspection30MaintDoor.monitoring.DoorOpen := "Safety.DataFromSafety".BA60jrPPLeftDoorForcedOpen OR "Safety.DataFromSafety".BA60jrPPLeftDoorNormalOpen;
   "OtherSafetyInterface".Inspection30MaintDoor.monitoring.DoorUnLock := "OtherSafetyInterface".Inspection30MaintDoor.monitoring.DoorOpen;
   "OtherSafetyInterface".Inspection30MaintDoor.monitoring.DoorClose := NOT "Safety.DataFromSafety".BA60jrPPLeftDoorForcedOpen AND NOT "Safety.DataFromSafety".BA60jrPPLeftDoorNormalOpen;
   "OtherSafetyInterface".Inspection30MaintDoor.monitoring.DoorLock := "OtherSafetyInterface".Inspection30MaintDoor.monitoring.DoorClose;
END_REGION

REGION Network 19: Inspection40Door Monitoring
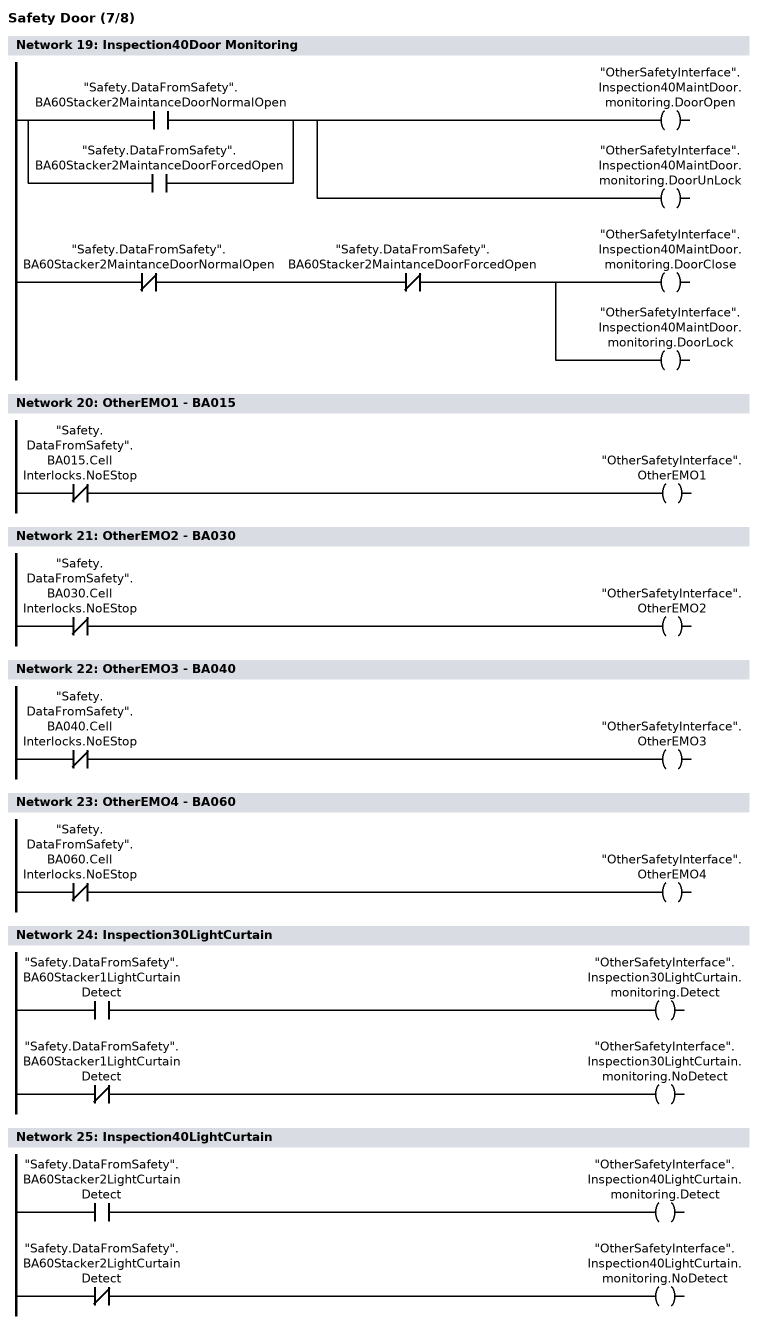
   RUNG wire#powerrail
      Contact( "Safety.DataFromSafety".BA60Stacker2MaintanceDoorNormalOpen )
      wire#w1
      Coil( "OtherSafetyInterface".Inspection40MaintDoor.monitoring.DoorOpen )
   END_RUNG
   RUNG wire#powerrail
      Contact( "Safety.DataFromSafety".BA60Stacker2MaintanceDoorForcedOpen )
   END_RUNG wire#w1
   RUNG wire#w1
      Coil( "OtherSafetyInterface".Inspection40MaintDoor.monitoring.DoorUnLock )
   END_RUNG
   RUNG wire#powerrail
      I_Contact( "Safety.DataFromSafety".BA60Stacker2MaintanceDoorNormalOpen )
      I_Contact( "Safety.DataFromSafety".BA60Stacker2MaintanceDoorForcedOpen )
      wire#w2
      Coil( "OtherSafetyInterface".Inspection40MaintDoor.monitoring.DoorClose )
   END_RUNG
   RUNG wire#w2
      Coil( "OtherSafetyInterface".Inspection40MaintDoor.monitoring.DoorLock )
   END_RUNG
   // the same network as SCL:
   "OtherSafetyInterface".Inspection40MaintDoor.monitoring.DoorOpen := "Safety.DataFromSafety".BA60Stacker2MaintanceDoorNormalOpen OR "Safety.DataFromSafety".BA60Stacker2MaintanceDoorForcedOpen;
   "OtherSafetyInterface".Inspection40MaintDoor.monitoring.DoorUnLock := "OtherSafetyInterface".Inspection40MaintDoor.monitoring.DoorOpen;
   "OtherSafetyInterface".Inspection40MaintDoor.monitoring.DoorClose := NOT "Safety.DataFromSafety".BA60Stacker2MaintanceDoorNormalOpen AND NOT "Safety.DataFromSafety".BA60Stacker2MaintanceDoorForcedOpen;
   "OtherSafetyInterface".Inspection40MaintDoor.monitoring.DoorLock := "OtherSafetyInterface".Inspection40MaintDoor.monitoring.DoorClose;
END_REGION

REGION Network 20: OtherEMO1 - BA015
   RUNG wire#powerrail
      I_Contact( "Safety.DataFromSafety".BA015.CellInterlocks.NoEStop )
      Coil( "OtherSafetyInterface".OtherEMO1 )
   END_RUNG
   // the same network as SCL:
   "OtherSafetyInterface".OtherEMO1 := NOT "Safety.DataFromSafety".BA015.CellInterlocks.NoEStop;
END_REGION

REGION Network 21: OtherEMO2 - BA030
   RUNG wire#powerrail
      I_Contact( "Safety.DataFromSafety".BA030.CellInterlocks.NoEStop )
      Coil( "OtherSafetyInterface".OtherEMO2 )
   END_RUNG
   // the same network as SCL:
   "OtherSafetyInterface".OtherEMO2 := NOT "Safety.DataFromSafety".BA030.CellInterlocks.NoEStop;
END_REGION

REGION Network 22: OtherEMO3 - BA040
   RUNG wire#powerrail
      I_Contact( "Safety.DataFromSafety".BA040.CellInterlocks.NoEStop )
      Coil( "OtherSafetyInterface".OtherEMO3 )
   END_RUNG
   // the same network as SCL:
   "OtherSafetyInterface".OtherEMO3 := NOT "Safety.DataFromSafety".BA040.CellInterlocks.NoEStop;
END_REGION

REGION Network 23: OtherEMO4 - BA060
   RUNG wire#powerrail
      I_Contact( "Safety.DataFromSafety".BA060.CellInterlocks.NoEStop )
      Coil( "OtherSafetyInterface".OtherEMO4 )
   END_RUNG
   // the same network as SCL:
   "OtherSafetyInterface".OtherEMO4 := NOT "Safety.DataFromSafety".BA060.CellInterlocks.NoEStop;
END_REGION

REGION Network 24: Inspection30LightCurtain
   RUNG wire#powerrail
      Contact( "Safety.DataFromSafety".BA60Stacker1LightCurtainDetect )
      Coil( "OtherSafetyInterface".Inspection30LightCurtain.monitoring.Detect )
   END_RUNG
   RUNG wire#powerrail
      I_Contact( "Safety.DataFromSafety".BA60Stacker1LightCurtainDetect )
      Coil( "OtherSafetyInterface".Inspection30LightCurtain.monitoring.NoDetect )
   END_RUNG
   // the same network as SCL:
   "OtherSafetyInterface".Inspection30LightCurtain.monitoring.Detect := "Safety.DataFromSafety".BA60Stacker1LightCurtainDetect;
   "OtherSafetyInterface".Inspection30LightCurtain.monitoring.NoDetect := NOT "Safety.DataFromSafety".BA60Stacker1LightCurtainDetect;
END_REGION

REGION Network 25: Inspection40LightCurtain
   RUNG wire#powerrail
      Contact( "Safety.DataFromSafety".BA60Stacker2LightCurtainDetect )
      Coil( "OtherSafetyInterface".Inspection40LightCurtain.monitoring.Detect )
   END_RUNG
   RUNG wire#powerrail
      I_Contact( "Safety.DataFromSafety".BA60Stacker2LightCurtainDetect )
      Coil( "OtherSafetyInterface".Inspection40LightCurtain.monitoring.NoDetect )
   END_RUNG
   // the same network as SCL:
   "OtherSafetyInterface".Inspection40LightCurtain.monitoring.Detect := "Safety.DataFromSafety".BA60Stacker2LightCurtainDetect;
   "OtherSafetyInterface".Inspection40LightCurtain.monitoring.NoDetect := NOT "Safety.DataFromSafety".BA60Stacker2LightCurtainDetect;
END_REGION

REGION Network 26: 30CathodeConveyorCover
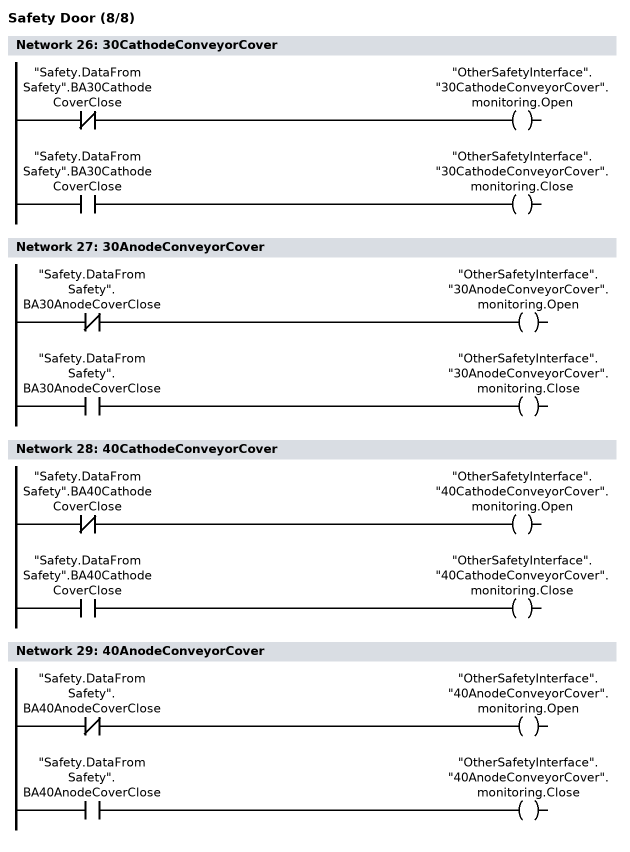
   RUNG wire#powerrail
      I_Contact( "Safety.DataFromSafety".BA30CathodeCoverClose )
      Coil( "OtherSafetyInterface"."30CathodeConveyorCover".monitoring.Open )
   END_RUNG
   RUNG wire#powerrail
      Contact( "Safety.DataFromSafety".BA30CathodeCoverClose )
      Coil( "OtherSafetyInterface"."30CathodeConveyorCover".monitoring.Close )
   END_RUNG
   // the same network as SCL:
   "OtherSafetyInterface"."30CathodeConveyorCover".monitoring.Open := NOT "Safety.DataFromSafety".BA30CathodeCoverClose;
   "OtherSafetyInterface"."30CathodeConveyorCover".monitoring.Close := "Safety.DataFromSafety".BA30CathodeCoverClose;
END_REGION

REGION Network 27: 30AnodeConveyorCover
   RUNG wire#powerrail
      I_Contact( "Safety.DataFromSafety".BA30AnodeCoverClose )
      Coil( "OtherSafetyInterface"."30AnodeConveyorCover".monitoring.Open )
   END_RUNG
   RUNG wire#powerrail
      Contact( "Safety.DataFromSafety".BA30AnodeCoverClose )
      Coil( "OtherSafetyInterface"."30AnodeConveyorCover".monitoring.Close )
   END_RUNG
   // the same network as SCL:
   "OtherSafetyInterface"."30AnodeConveyorCover".monitoring.Open := NOT "Safety.DataFromSafety".BA30AnodeCoverClose;
   "OtherSafetyInterface"."30AnodeConveyorCover".monitoring.Close := "Safety.DataFromSafety".BA30AnodeCoverClose;
END_REGION

REGION Network 28: 40CathodeConveyorCover
   RUNG wire#powerrail
      I_Contact( "Safety.DataFromSafety".BA40CathodeCoverClose )
      Coil( "OtherSafetyInterface"."40CathodeConveyorCover".monitoring.Open )
   END_RUNG
   RUNG wire#powerrail
      Contact( "Safety.DataFromSafety".BA40CathodeCoverClose )
      Coil( "OtherSafetyInterface"."40CathodeConveyorCover".monitoring.Close )
   END_RUNG
   // the same network as SCL:
   "OtherSafetyInterface"."40CathodeConveyorCover".monitoring.Open := NOT "Safety.DataFromSafety".BA40CathodeCoverClose;
   "OtherSafetyInterface"."40CathodeConveyorCover".monitoring.Close := "Safety.DataFromSafety".BA40CathodeCoverClose;
END_REGION

REGION Network 29: 40AnodeConveyorCover
   RUNG wire#powerrail
      I_Contact( "Safety.DataFromSafety".BA40AnodeCoverClose )
      Coil( "OtherSafetyInterface"."40AnodeConveyorCover".monitoring.Open )
   END_RUNG
   RUNG wire#powerrail
      Contact( "Safety.DataFromSafety".BA40AnodeCoverClose )
      Coil( "OtherSafetyInterface"."40AnodeConveyorCover".monitoring.Close )
   END_RUNG
   // the same network as SCL:
   "OtherSafetyInterface"."40AnodeConveyorCover".monitoring.Open := NOT "Safety.DataFromSafety".BA40AnodeCoverClose;
   "OtherSafetyInterface"."40AnodeConveyorCover".monitoring.Close := "Safety.DataFromSafety".BA40AnodeCoverClose;
END_REGION
END_FUNCTION
